{attribute 'reflection'}
FUNCTION_BLOCK FB_EncoderInput EXTENDS FB_EncoderBase
VAR_INPUT
END_VAR
VAR_OUTPUT
END_VAR
VAR
	iCounterValue 	AT%I*	: UDINT ;
	iDataError		AT%I*	: BOOL  ;	
	iFrameError		AT%I*	: BOOL  ;
	iPowerFailure	AT%I*	: BOOL  ; 
	iSyncError		AT%I*	: BOOL  ;
	
	nScaledValue		: LREAL ; // Only scaled value for internal use
	nValueWithOffset	: LREAL ; // scaled value with added offset
	fOldPos				: LREAL ; // Old position
	
END_VAR

// ====== Check device status ======
	CheckBoxStatus();

// ====== Scale Output value ======
	nScaledValue := UDINT_TO_LREAL(iCounterValue) / fPulsesPerUnit ;

// ====== Invert ======
	IF bIcfInverted THEN 
		nScaledValue := nScaledValue * -1;
	END_IF
	
// ====== Add offset ======= 
	nValueWithOffset := nScaledValue + fOffset ;
	
// ====== Caclulate velocity =====
	IF Sys_Variables.Pulse100ms THEN 
		nVelocity 	:= (nOutPosition - fOldPos) * 10 ;
		fOldPos		:= nOutPosition;
	END_IF
	
// ====== Set Outputs =======
	nOutPosition 	:= nValueWithOffset ;
	nOutRaw			:= iCounterValue	;

METHOD PRIVATE CheckBoxStatus : BOOL
VAR_INPUT
END_VAR
IF iDataError THEN 
	stFault.Active 			:= TRUE ;
	stFault.Discription		:= CONCAT(sName, ' Encoder Data error');
	stFault.MessageNumber	:= E_MessageNumbers.FF_ComunicationFault;
	stFault.FaultType		:= E_FaultTypes.FF;
ELSIF iFrameError THEN 
	stFault.Active 			:= TRUE ;
	stFault.Discription		:= CONCAT(sName, ' Encoder frame error');
	stFault.MessageNumber	:= E_MessageNumbers.FF_ComunicationFault;
	stFault.FaultType		:= E_FaultTypes.FF;
ELSIF iPowerFailure THEN 
	stFault.Active 			:= TRUE ;
	stFault.Discription		:= CONCAT(sName, ' Encoder Power failure');
	stFault.MessageNumber	:= E_MessageNumbers.FF_ComunicationFault;
	stFault.FaultType		:= E_FaultTypes.FF;
ELSIF iSyncError THEN 
	stFault.Active 			:= TRUE ;
	stFault.Discription		:= CONCAT(sName, ' Encoder synchronisation error');
	stFault.MessageNumber	:= E_MessageNumbers.FF_ComunicationFault;
	stFault.FaultType		:= E_FaultTypes.FF;
END_IF
END_METHOD

METHOD PUBLIC FastTask : BOOL
VAR_INPUT
END_VAR
END_METHOD

END_FUNCTION_BLOCK

(* stored: Version 1.1.0.1, ProductVersion 3.1.4024.5
   POU FB_EncoderInput: Id {0f518a76-74dc-4426-927f-5208a6bc0566}, SpecialFunc None
   Method CheckBoxStatus: Id {955108e9-c9df-0ec1-0ba8-cf8484910c33}
   Method FastTask: Id {2447dce7-4abc-4c3e-b487-bf649a6d099a} *)
